Fanuc KAREL source: kt00058.KL

-- PROVISIONAL review KL for V940-1; original PC SHA256 2d3f6e958dd24b34faf6159f1d5e388e13d8437a004d816e487401c1f6dd3077
-- Incomplete behavior may be omitted. Consult companion uncertainty JSON. Do not deploy.
PROGRAM KT00058
%NOLOCKGROUP
VAR
  I2 : INTEGER
  OUT : REAL
-- UNRESOLVED_DECL H1 type=002017
BEGIN
  -- V9_ZERO_TABLE_METADATA_HINT layout=0001; no indexed target words; source/name/runtime held
  -- UNRESOLVED_PC offsets 5-19; opcodes 2E,22,9D,33,B4
  -- UNRESOLVED_PC offsets 24-35; opcodes 2E,23
  -- UNRESOLVED_PC offsets 40-63; opcodes 22,9D,33,B3,21,53,64,23
  -- UNRESOLVED_PC offsets 68-72; opcodes 7F
END KT00058
